(* Logix 5000 project; controller CarbonScout_MK6 vendor 1 type 14 code 154 rev 32.11; software revision 32.00; part 5 of 17 *)
(* tags used below, declared in another part *)
   Inp_OpenLS : BOOL;   // Valve Open Limit Switch 1=confirmed OPEN
   Inp_ClosedLS : BOOL;   // Valve Closed Limit Switch 1=confirmed CLOSED
   Inp_PermOK : BOOL;   // 1=Permissives OK, Valve can energize
   Inp_NBPermOK : BOOL;   // 1=Non-Bypassable Permissives OK, valve can energize
   Inp_IntlkOK : BOOL;   // 1=Interlocks OK, valve can energize
   Inp_NBIntlkOK : BOOL;   // 1=Non-Bypassable Interlocks OK, valve can energize
   Inp_IOFault : BOOL;   // Input Communication Status 0=OK, 1=fail
   Inp_Sim : BOOL;   // 1=Simulate working valve; 0=Open/Close/ Monitor actual valve
   Inp_OvrdCmd : DINT;   // Override Mode Command: 0=None, 1=Close, 2=Open
   Inp_Reset : BOOL;   // 1=Reset all fault conditions and latched Alarms
   Cfg_FailOpen : BOOL;   // 1=Fail Open (energize to close), 0=Fail Closed (energize to open)
   Cfg_HasOpenLS : BOOL;   // 1=Valve provides an Open Limit Switch signal
   Cfg_HasClosedLS : BOOL;   // 1=Valve provides a Closed Limit Switch signal
   Cfg_UseOpenLS : BOOL;   // 1=Valve Open LS should be used for failure checking
   Cfg_UseClosedLS : BOOL;   // 1=Valve Closed LS should be used for failure checking
   Cfg_LSFail : BOOL;   // 1=both switches ON=fail, 0=both switches OFF=fail
   Cfg_PCmdClear : ALIAS FOR Mode.Cfg_PCmdClear;
   Cfg_OCmdResets : BOOL;   // 1=New Oper valve cmd. resets fault, 0=reset req'd to clear fault
   Cfg_ShedOnFullStall : BOOL;   // 1=Stop Valve and Alarm on Full Stall; 0=Alarm only on Full Stall
   Cfg_ShedOnTransitStall : BOOL;   // 1=Stop Valve and Alarm on Transit Stall; 0=Alarm only on Transit Stall
   Cfg_ShedOnIOFault : BOOL;   // 1=Stop Valve and Alarm on I/O Fault; 0=Alarm only on I/O Fault
   Cfg_OvrdPermIntlk : BOOL;   // 1=Override ignores Bypassable Perm/ Intlk; 0=always use Perm/Intlk
   Cfg_SimFdbkT : DINT;   // Delay to echo back of Open/Closed status when in Simulation (sec)
   Cfg_FullStallT : DINT;   // After command, time with no motion before Fault (sec)
   Cfg_TransitStallT : DINT;   // After command, time to reach position before fault (sec)
   PSet_Owner : DINT;   // Program Owner Request ID (non-zero) or Release (zero)
   PCmd_Open : BOOL;   // Program Command to Open Valve
   PCmd_Close : BOOL;   // Program Command to Close Valve
   PCmd_Reset : BOOL;   // Program Command to Reset all Alarms requiring Reset
   PCmd_FullStallAck : ALIAS FOR FullStall.PCmd_Ack;   // Program Command to Acknowledge Full Stall Alarm
   PCmd_TransitStallAck : ALIAS FOR TransitStall.PCmd_Ack;   // Program Command to Acknowledge Transit Stall Alarm
   PCmd_IntlkTripAck : ALIAS FOR IntlkTrip.PCmd_Ack;   // Program Command to Acknowledge Interlock Trip Alarm
   PCmd_IOFaultAck : ALIAS FOR IOFault.PCmd_Ack;   // Program Command to Acknowledge I/O Fault Alarm
   OCmd_Open : BOOL;   // Operator Command to Open Valve
   OCmd_Close : BOOL;   // Operator Command to Close Valve
   OCmd_Bypass : BOOL;   // Operator Command to Bypass all Bypassable Interlocks and Permissives
   OCmd_Check : BOOL;   // Operator Command to Check (not bypass) all Interlocks and Permissives
   MCmd_Disable : BOOL;   // Maintenance Command to Disable Valve
   MCmd_Enable : BOOL;   // Maintenance Command to Enable (allow to energize) Valve
   OCmd_Reset : BOOL;   // Operator Command to Reset all Alarms requiring Reset
   OCmd_ResetAckAll : BOOL;   // Operator Command to Reset all Alarms and latched Shed conditions
   Out : BOOL;   // 1=Energize Valve Solenoid
   SrcQ_IO : DINT;   // Source and Quality of primary I/O (enumeration)
   SrcQ : DINT;   // Source and Quality of primary Val/Sts (enumeration)
   Val_Cmd : DINT;   // Device Command 0=None, 1=Close, 2=Open
   Val_Fdbk : DINT;   // Device Feedback 0=Moving, 1=Closed, 2=Opened, 3=Limit Switch Failure
   Val_Sts : DINT;   // Device Confirmed Sts 0=? 1=Closed 2=Open 5=Closing, 6=Opening, 33=Disabled
   Val_Fault : DINT;   // Device Fault Status 0=None, 16=Transit Stall, 17 = Full Stall, 32=I/O Fault, 34=Config Error
   Val_Owner : DINT;   // Current Object Owner ID (0=not owned)
   Sts_Closed : BOOL;   // 1=Valve requested to Close and is confirmed Closed
   Sts_Opening : BOOL;   // 1=Valve requested to open and awaiting open feedback
   Sts_Opened : BOOL;   // 1=Valve requested to open and is confirmed Opened
   Sts_Closing : BOOL;   // 1=Valve requested to Close and awaiting Closed feedback
   Sts_Available : BOOL;   // 1=Valve available for control by automation (Prog)
   Sts_Bypass : BOOL;   // 1=Bypassable Interlocks and Permissives are Bypassed
   Sts_BypActive : BOOL;   // 1=Bypassing Active (Bypassed or Maintenance)
   Sts_Disabled : BOOL;   // 1=Valve is Disabled
   Sts_LSFail : BOOL;   // 1=Limit Switch Overlap Failure
   Sts_NotRdy : BOOL;   // 1=Device Not Ready, see detail bits for reason
   Nrdy_Disabled : BOOL;   // 1=Device Not Ready: Device Disabled by Maintenance
   Nrdy_CfgErr : BOOL;   // 1=Device Not Ready: Configuration Error
   Nrdy_Intlk : BOOL;   // 1=Device Not Ready: Interlock Not OK
   Nrdy_Perm : BOOL;   // 1=Device Not Ready: Permissive Not OK
   Nrdy_Fail : BOOL;   // 1=Device Not Ready: Device Failure (Shed Requires Reset)
   Nrdy_IOFault : BOOL;   // 1=Device Not Ready: I/O Fault (Shed Requires Reset)
   Nrdy_NoMode : BOOL;   // 1=Device Not Ready: Device Logic Disabled / NO Mode
   Sts_MaintByp : BOOL;   // 1=A Maintenance Bypass is Active, display icon
   Sts_Err : BOOL;   // 1=Error in Config: see detail bits for reason
   Err_Timer : BOOL;   // 1=Error in Config: Invalid Check Time (use 0 to 2147483)
   Err_Sim : BOOL;   // 1=Error in Config: Invalid Simulation Time (use 0 to 2147483)
   Err_Alarm : BOOL;   // 1=Error in Config: Alarm Min On Time, Shelf Time, Severity
   Sts_Hand : ALIAS FOR Mode.Sts_Hand;
   Sts_Maint : ALIAS FOR Mode.Sts_Maint;
   Sts_Ovrd : ALIAS FOR Mode.Sts_Ovrd;
   Sts_Prog : ALIAS FOR Mode.Sts_Prog;
   Sts_Oper : ALIAS FOR Mode.Sts_Oper;
   Sts_FullStall : ALIAS FOR FullStall.Inp;   // 1=Valve Full Stall (failed to move at all)
   Sts_TransitStall : ALIAS FOR TransitStall.Inp;   // 1=Valve Transit Stall (did not reach target position)
   Sts_IntlkTrip : ALIAS FOR IntlkTrip.Inp;   // 1=Valve de-energized by an Interlock NOT OK
   Sts_IOFault : ALIAS FOR IOFault.Inp;   // I/O Comm Fault Status (0=OK, 1=Bad)
   Rdy_Open : BOOL;   // 1=Ready to receive OCmd_Open (enables HMI button)
   Rdy_Close : BOOL;   // 1=Ready to receive OCmd_Close (enables HMI button)
   Rdy_Bypass : BOOL;   // 1=Ready to receive OCmd_Bypass (enables HMI button)
   Rdy_Check : BOOL;   // 1=Ready to receive OCmd_Check (enables HMI button)
   Rdy_Disable : BOOL;   // 1=Ready to receive MCmd_Disable (enables HMI button)
   Rdy_Enable : BOOL;   // 1=Ready to receive MCmd_Enable (enables HMI button)
   P_ValveSO : BOOL;   // Unique Parameter Name for auto - discovery
   Mode : P_Mode;   // Valve Mode Selection
   IOFault : P_Alarm;   // I/O Fault Alarm
   IntlkTrip : P_Alarm;   // Interlock Trip Alarm
   TransitStall : P_Alarm;   // Valve Transit Stall (moved but did not reach target) Alarm
   FullStall : P_Alarm;   // Valve Full Stall (did not move) Alarm
   Cfg_Tag : STRING_12;   // Tagname for display on HMI
   Wrk_Open : BOOL;   // 1=Requested to OPEN Valve, 0=Requested to CLOSE Valve
   Wrk_SimOpenT : TIMER;   // Simulation Delay until Opened
   Wrk_SimCloseT : TIMER;   // Simulation Delay until Closed
   Wrk_OpenFdbk : BOOL;   // 1=LS Feedback shows valve confirmed open
   Wrk_Bypass : BOOL;   // Internal Bypassable Permissives and Interlocks are Bypassed flag
   Wrk_Disabled : BOOL;   // Internal Valve is Disabled
   Wrk_ClosedFdbk : BOOL;   // 1=LS Feedback shows valve confirmed closed
   Wrk_TransitStallT : TIMER;   // Timer for Transit Stall Check
   Wrk_FullStallT : TIMER;   // Timer for Full Stall Check
   Wrk_Sts : DINT;   // Buffer for building Val_Sts
   Wrk_SrcQ : DINT;   // Register for building Source / Quality enumeration
   Wrk_Fault : DINT;   // Buffer for building Val_Fault
   Wrk_Cmd : DINT;   // Buffer for building Val_Cmd
   Wrk_SimOpenLS : BOOL;   // Simulated valve Open Limit Switch
   Wrk_SimClosedLS : BOOL;   // Simulated valve Closed Limit Switch
   Wrk_NotRdy : BOOL;   // Device Not Ready conditions excluding shed latches
   Wrk_NoLongerSim : BOOL;   // Switched from Simulated to Real Valve this scan
   Simulation : DINT;
   test : DINT;
(* P_ValveSO, continued *)

ROUTINE Logic   (* ladder *)
// Normal Scan: control / monitor solenoid-operated valve
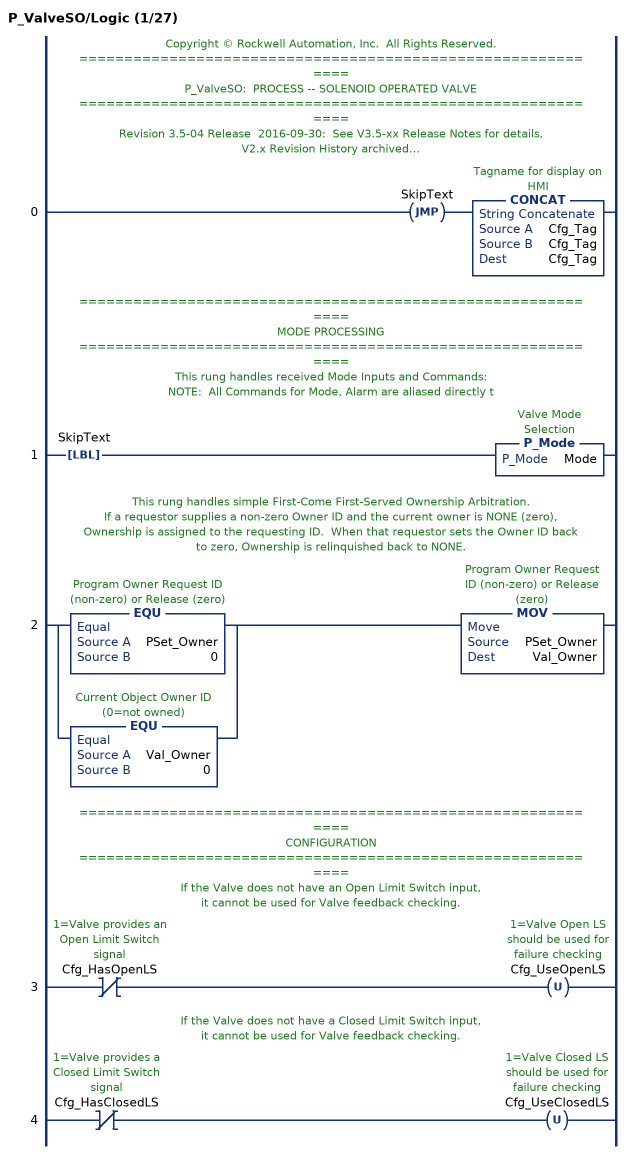
   // Copyright © Rockwell Automation, Inc.  All Rights Reserved.
   // ============================================================
   // P_ValveSO:  PROCESS -- SOLENOID OPERATED VALVE
   // ============================================================
   // Revision 3.5-04 Release  2016-09-30:  See V3.5-xx Release Notes for details.
   // V2.x Revision History archived.
   // V3.0-00  2013-06-30:  Added Inf_Lib. Using P_Alarm, P_Mode V3.0.
   // V3.0-01  2013-07-31:  Modified Parameter descriptions only.
   // V3.0-02  2013-09-03:  Modified Parameter descriptions only.
   // V3.0-03  2013-10-30:  Prescan code modified for proper powerup state.
   // Corrected Parameter descriptions and default
   // configuration values for alarms.
   // V3.0-04  2014-01-22:  Corrected Parameter Description for Val_Sts.
   // V3.1-00  2014-07-08:  Modified to use P_Alarm, P_Mode V3.1. Added Not
   // Ready reason bits (Nrdy_Xxxxx), source/quality values (SrcQ).
   // Modified to consistently use alias tag names.
   // V3.1-01  2014-09-03:  Exposed stall timers ACC/PRE (read-only). Corrections to
   // Nrdy_ trip and reset logic. Using P_Alarm, P_Mode V3.1-01.
   // V3.1-02  2014-09-30:  Unchanged, but using P_Alarm V3.1-02.
   // V3.5-01  2016-01-29:  Unchanged, but using P_Alarm V3.5.01.
   // V3.5-04  2016-09-30: Modified to align with actual device state on transition
   // from Sim to real valve.
   // ============================================================
   // This Instruction controls and monitors a single solenoid operated
   // valve (typ. two position: opened, closed) and provides:
   // *  Support for fail open (energize to close) and fail closed (energize to open, default) valves
   // *  Monitoring of limit switch feedback, display of actual valve status
   // *  Detection of failure to move (full stall), failure to reach position (transit stall)
   // *  Monitoring of Permissive conditions to allow energizing
   // *  Monitoring of Interlock conditions to de-energize
   // *  Simulation, providing feedback of a working valve while disabling outputs
   // *  Monitoring of I/O communication faults
   // *  Alarms for Full Stall, Transit Stall, Interlock Trip, I/O Fault
   // *  "Available" status for use by automation logic to know whether valve
   //       can be controlled by other objects.
   // Modes are provided by a P_Mode AOI instance.
   // Alarms are provided by P_Alarm AOI instances.
   // Modes of operation: Operator, Program, Override, Maintenance, Hand
   // ============================================================
   // SHOW LOCAL STRINGS
   // ============================================================
   // The STRINGs containing the text associated with each instance of this
   // instruction cannot be Input or Output Parameters, because STRINGs are not
   //  'atomic' types. (Inputs and Outputs must be SINT, INT, DINT, REAL, or BOOL.)
   // In order to make it easier to find and configure these STRINGs, this rung
   // was added.  THE JMP (and the LBL on the following rung)
   // MUST NOT BE REMOVED!!!
   // To view the STRINGs, go to the instruction instance (in LD or FBD), RIGHT-click
   // to bring up the context menu and select "Open Instruction Logic".
   // This rung will appear with the STRING values for the selected instance.
   // You may double-click the STRING values here to modify them as well.
   0: JMP(SkipText)CONCAT(Cfg_Tag,Cfg_Tag,Cfg_Tag);
   // ============================================================
   // MODE PROCESSING
   // ============================================================
   // This rung handles received Mode Inputs and Commands:
   // NOTE:  All Commands for Mode, Alarm are aliased directly t
   1: LBL(SkipText)P_Mode(Mode);
   // This rung handles simple First-Come First-Served Ownership Arbitration.
   // If a requestor supplies a non-zero Owner ID and the current owner is NONE (zero),
   // Ownership is assigned to the requesting ID.  When that requestor sets the Owner ID back
   // to zero, Ownership is relinquished back to NONE.
   2: [EQU(PSet_Owner,0) ,EQU(Val_Owner,0) ]MOV(PSet_Owner,Val_Owner);
   // ============================================================
   // CONFIGURATION
   // ============================================================
   // If the Valve does not have an Open Limit Switch input,
   // it cannot be used for Valve feedback checking.
   3: XIO(Cfg_HasOpenLS)OTU(Cfg_UseOpenLS);
   // If the Valve does not have a Closed Limit Switch input,
   // it cannot be used for Valve feedback checking.
   4: XIO(Cfg_HasClosedLS)OTU(Cfg_UseClosedLS);
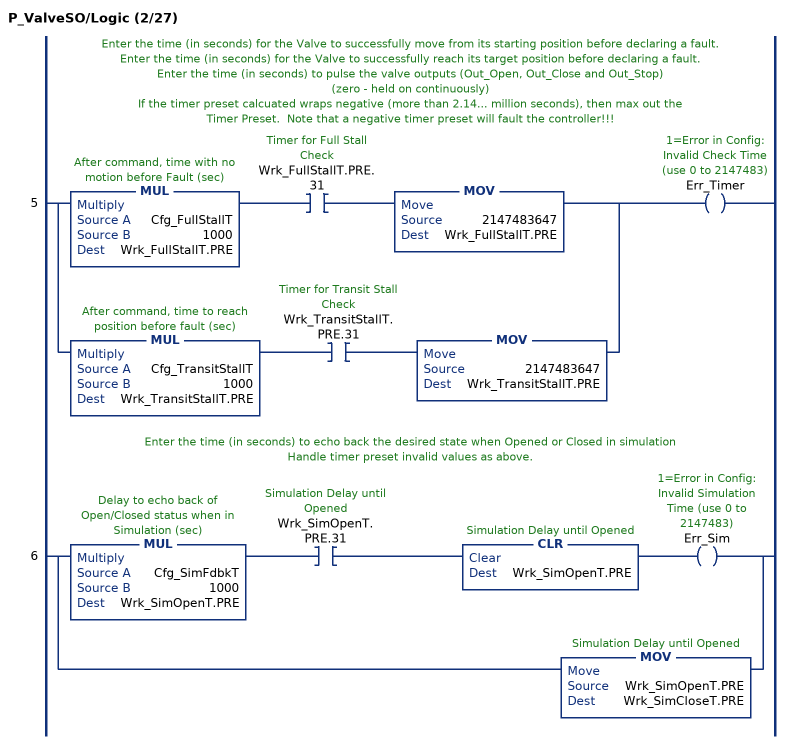
   // Enter the time (in seconds) for the Valve to successfully move from its starting position before declaring a fault.
   // Enter the time (in seconds) for the Valve to successfully reach its target position before declaring a fault.
   // Enter the time (in seconds) to pulse the valve outputs (Out_Open, Out_Close and Out_Stop)
   // (zero - held on continuously)
   // If the timer preset calcuated wraps negative (more than 2.14... million seconds), then max out the
   // Timer Preset.  Note that a negative timer preset will fault the controller!!!
   5: [MUL(Cfg_FullStallT,1000,Wrk_FullStallT.PRE) XIC(Wrk_FullStallT.PRE.31) MOV(2147483647,Wrk_FullStallT.PRE) ,MUL(Cfg_TransitStallT,1000,Wrk_TransitStallT.PRE) XIC(Wrk_TransitStallT.PRE.31) MOV(2147483647,Wrk_TransitStallT.PRE) ]OTE(Err_Timer);
   // Enter the time (in seconds) to echo back the desired state when Opened or Closed in simulation
   // Handle timer preset invalid values as above.
   6: [MUL(Cfg_SimFdbkT,1000,Wrk_SimOpenT.PRE) XIC(Wrk_SimOpenT.PRE.31) CLR(Wrk_SimOpenT.PRE) OTE(Err_Sim) ,MOV(Wrk_SimOpenT.PRE,Wrk_SimCloseT.PRE) ];
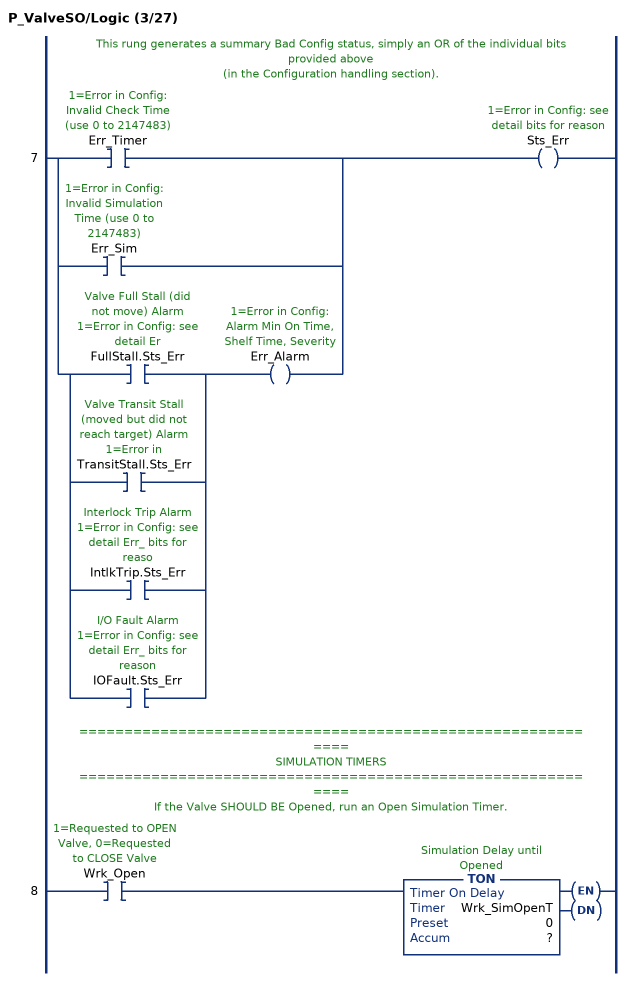
   // This rung generates a summary Bad Config status, simply an OR of the individual bits provided above
   // (in the Configuration handling section).
   7: [XIC(Err_Timer) ,XIC(Err_Sim) ,[XIC(FullStall.Sts_Err) ,XIC(TransitStall.Sts_Err) ,XIC(IntlkTrip.Sts_Err) ,XIC(IOFault.Sts_Err) ] OTE(Err_Alarm) ]OTE(Sts_Err);
   // ============================================================
   // SIMULATION TIMERS
   // ============================================================
   // If the Valve SHOULD BE Opened, run an Open Simulation Timer.
   8: XIC(Wrk_Open)TON(Wrk_SimOpenT,?,?);
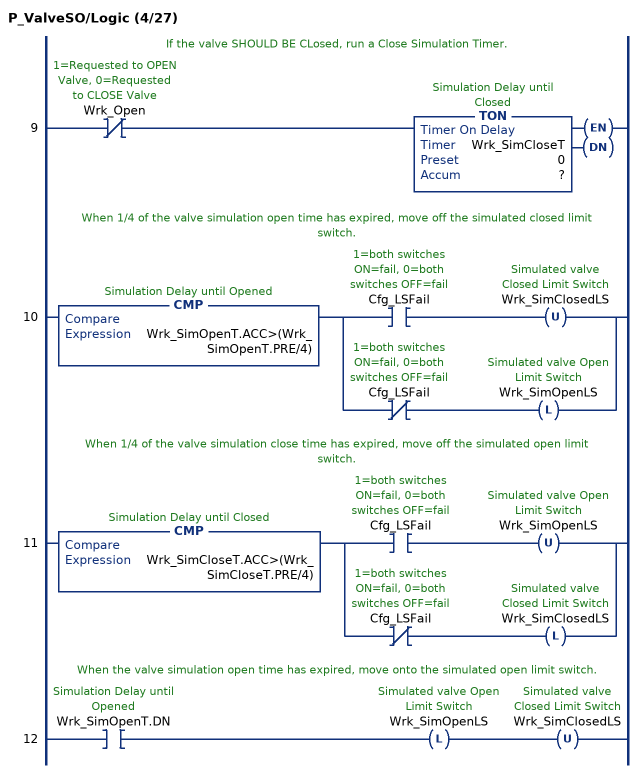
   // If the valve SHOULD BE CLosed, run a Close Simulation Timer.
   9: XIO(Wrk_Open)TON(Wrk_SimCloseT,?,?);
   // When 1/4 of the valve simulation open time has expired, move off the simulated closed limit switch.
   10: CMP(Wrk_SimOpenT.ACC>(Wrk_SimOpenT.PRE/4))[XIC(Cfg_LSFail) OTU(Wrk_SimClosedLS) ,XIO(Cfg_LSFail) OTL(Wrk_SimOpenLS) ];
   // When 1/4 of the valve simulation close time has expired, move off the simulated open limit switch.
   11: CMP(Wrk_SimCloseT.ACC>(Wrk_SimCloseT.PRE/4))[XIC(Cfg_LSFail) OTU(Wrk_SimOpenLS) ,XIO(Cfg_LSFail) OTL(Wrk_SimClosedLS) ];
   // When the valve simulation open time has expired, move onto the simulated open limit switch.
   12: XIC(Wrk_SimOpenT.DN)OTL(Wrk_SimOpenLS)OTU(Wrk_SimClosedLS);
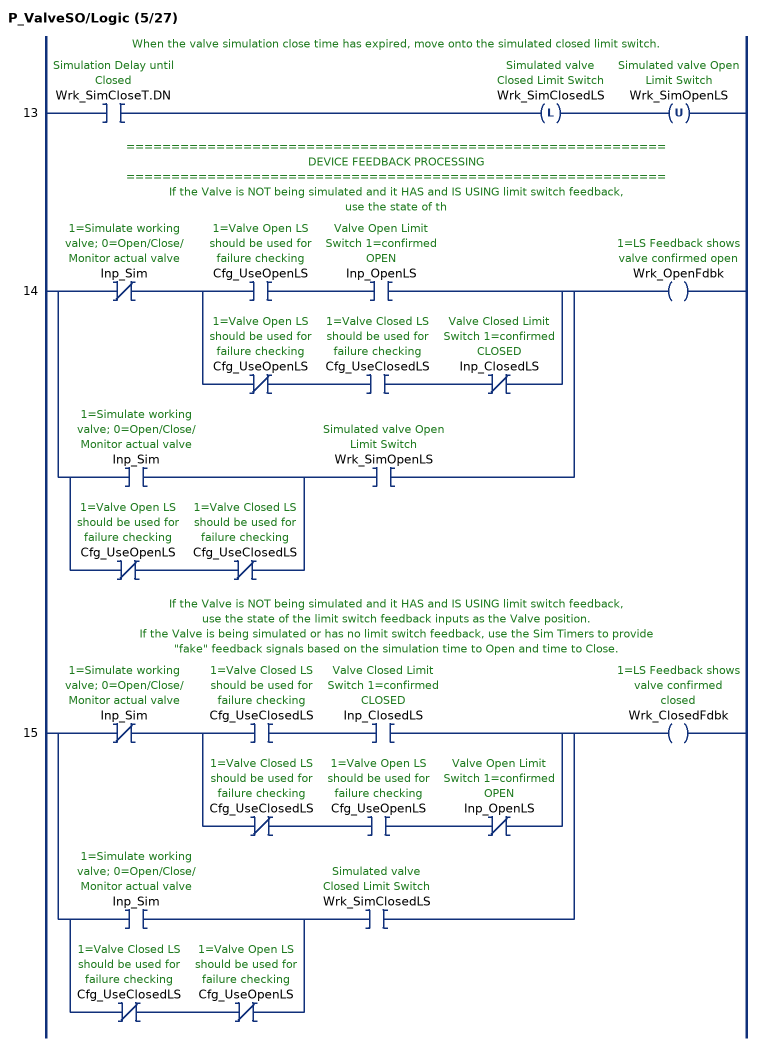
   // When the valve simulation close time has expired, move onto the simulated closed limit switch.
   13: XIC(Wrk_SimCloseT.DN)OTL(Wrk_SimClosedLS)OTU(Wrk_SimOpenLS);
   // ============================================================
   // DEVICE FEEDBACK PROCESSING
   // ============================================================
   // If the Valve is NOT being simulated and it HAS and IS USING limit switch feedback,
   // use the state of th
   14: [XIO(Inp_Sim) [XIC(Cfg_UseOpenLS) XIC(Inp_OpenLS) ,XIO(Cfg_UseOpenLS) XIC(Cfg_UseClosedLS) XIO(Inp_ClosedLS) ] ,[XIC(Inp_Sim) ,XIO(Cfg_UseOpenLS) XIO(Cfg_UseClosedLS) ] XIC(Wrk_SimOpenLS) ]OTE(Wrk_OpenFdbk);
   // If the Valve is NOT being simulated and it HAS and IS USING limit switch feedback,
   // use the state of the limit switch feedback inputs as the Valve position.
   // If the Valve is being simulated or has no limit switch feedback, use the Sim Timers to provide
   // "fake" feedback signals based on the simulation time to Open and time to Close.
   15: [XIO(Inp_Sim) [XIC(Cfg_UseClosedLS) XIC(Inp_ClosedLS) ,XIO(Cfg_UseClosedLS) XIC(Cfg_UseOpenLS) XIO(Inp_OpenLS) ] ,[XIC(Inp_Sim) ,XIO(Cfg_UseClosedLS) XIO(Cfg_UseOpenLS) ] XIC(Wrk_SimClosedLS) ]OTE(Wrk_ClosedFdbk);
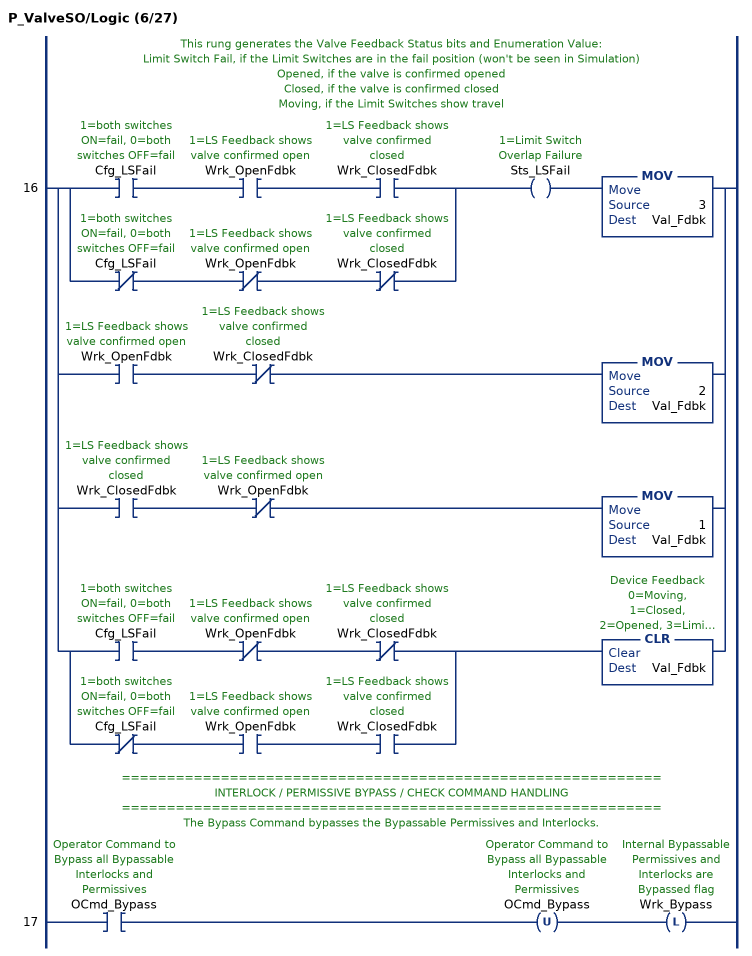
   // This rung generates the Valve Feedback Status bits and Enumeration Value:
   // Limit Switch Fail, if the Limit Switches are in the fail position (won't be seen in Simulation)
   // Opened, if the valve is confirmed opened
   // Closed, if the valve is confirmed closed
   // Moving, if the Limit Switches show travel
   16: [[XIC(Cfg_LSFail) XIC(Wrk_OpenFdbk) XIC(Wrk_ClosedFdbk) ,XIO(Cfg_LSFail) XIO(Wrk_OpenFdbk) XIO(Wrk_ClosedFdbk) ] OTE(Sts_LSFail) MOV(3,Val_Fdbk) ,XIC(Wrk_OpenFdbk) XIO(Wrk_ClosedFdbk) MOV(2,Val_Fdbk) ,XIC(Wrk_ClosedFdbk) XIO(Wrk_OpenFdbk) MOV(1,Val_Fdbk) ,[XIC(Cfg_LSFail) XIO(Wrk_OpenFdbk) XIO(Wrk_ClosedFdbk) ,XIO(Cfg_LSFail) XIC(Wrk_OpenFdbk) XIC(Wrk_ClosedFdbk) ] CLR(Val_Fdbk) ];
   // ============================================================
   // INTERLOCK / PERMISSIVE BYPASS / CHECK COMMAND HANDLING
   // ============================================================
   // The Bypass Command bypasses the Bypassable Permissives and Interlocks.
   17: XIC(OCmd_Bypass)OTU(OCmd_Bypass)OTL(Wrk_Bypass);
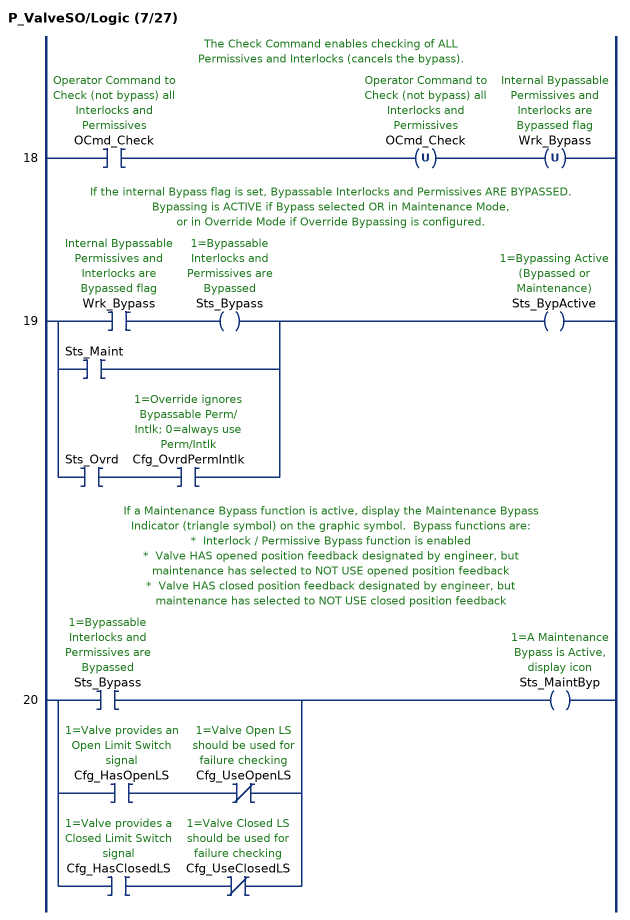
   // The Check Command enables checking of ALL
   // Permissives and Interlocks (cancels the bypass).
   18: XIC(OCmd_Check)OTU(OCmd_Check)OTU(Wrk_Bypass);
   // If the internal Bypass flag is set, Bypassable Interlocks and Permissives ARE BYPASSED.
   // Bypassing is ACTIVE if Bypass selected OR in Maintenance Mode,
   // or in Override Mode if Override Bypassing is configured.
   19: [XIC(Wrk_Bypass) OTE(Sts_Bypass) ,XIC(Sts_Maint) ,XIC(Sts_Ovrd) XIC(Cfg_OvrdPermIntlk) ]OTE(Sts_BypActive);
   // If a Maintenance Bypass function is active, display the Maintenance Bypass
   // Indicator (triangle symbol) on the graphic symbol.  Bypass functions are:
   // *  Interlock / Permissive Bypass function is enabled
   // *  Valve HAS opened position feedback designated by engineer, but
   // maintenance has selected to NOT USE opened position feedback
   // *  Valve HAS closed position feedback designated by engineer, but
   // maintenance has selected to NOT USE closed position feedback
   20: [XIC(Sts_Bypass) ,XIC(Cfg_HasOpenLS) XIO(Cfg_UseOpenLS) ,XIC(Cfg_HasClosedLS) XIO(Cfg_UseClosedLS) ]OTE(Sts_MaintByp);
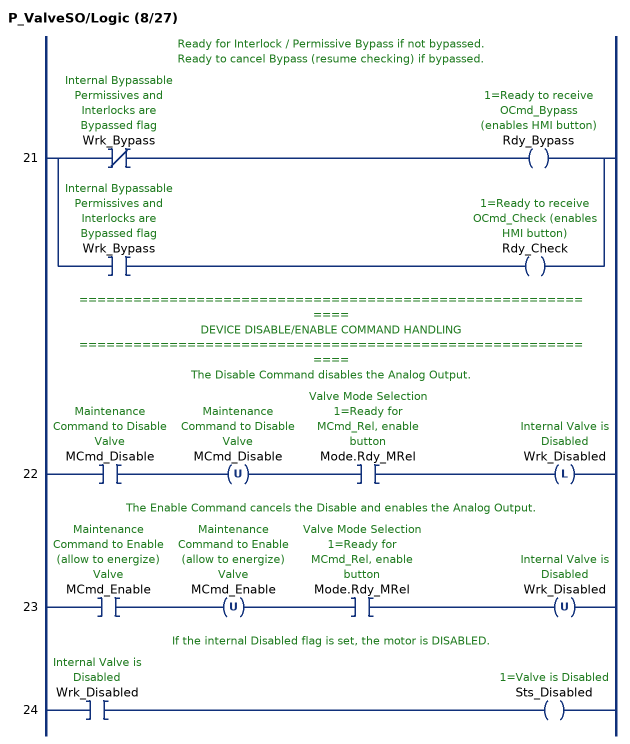
   // Ready for Interlock / Permissive Bypass if not bypassed.
   // Ready to cancel Bypass (resume checking) if bypassed.
   21: [XIO(Wrk_Bypass) OTE(Rdy_Bypass) ,XIC(Wrk_Bypass) OTE(Rdy_Check) ];
   // ============================================================
   // DEVICE DISABLE/ENABLE COMMAND HANDLING
   // ============================================================
   // The Disable Command disables the Analog Output.
   22: XIC(MCmd_Disable)OTU(MCmd_Disable)XIC(Mode.Rdy_MRel)OTL(Wrk_Disabled);
   // The Enable Command cancels the Disable and enables the Analog Output.
   23: XIC(MCmd_Enable)OTU(MCmd_Enable)XIC(Mode.Rdy_MRel)OTU(Wrk_Disabled);
   // If the internal Disabled flag is set, the motor is DISABLED.
   24: XIC(Wrk_Disabled)OTE(Sts_Disabled);
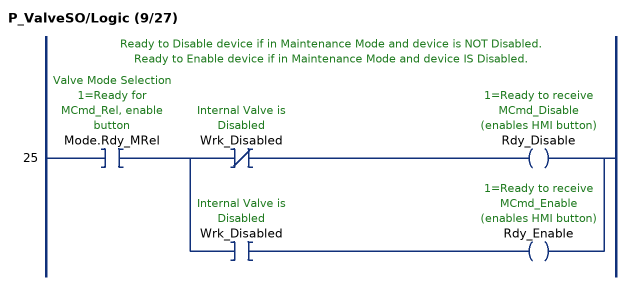
   // Ready to Disable device if in Maintenance Mode and device is NOT Disabled.
   // Ready to Enable device if in Maintenance Mode and device IS Disabled.
   25: XIC(Mode.Rdy_MRel)[XIO(Wrk_Disabled) OTE(Rdy_Disable) ,XIC(Wrk_Disabled) OTE(Rdy_Enable) ];
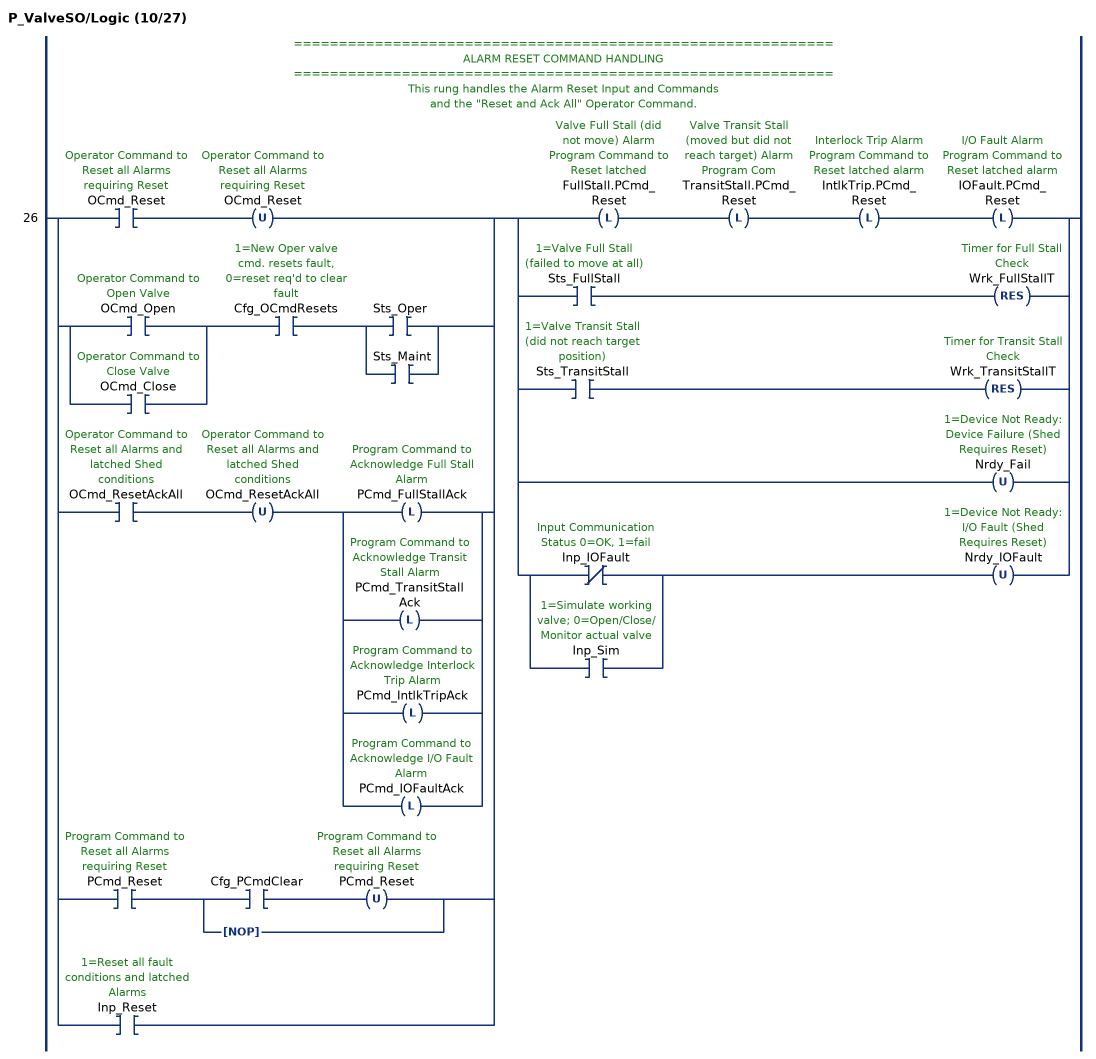
   // ============================================================
   // ALARM RESET COMMAND HANDLING
   // ============================================================
   // This rung handles the Alarm Reset Input and Commands
   // and the "Reset and Ack All" Operator Command.
   26: [XIC(OCmd_Reset) OTU(OCmd_Reset) ,[XIC(OCmd_Open) ,XIC(OCmd_Close) ] XIC(Cfg_OCmdResets) [XIC(Sts_Oper) ,XIC(Sts_Maint) ] ,XIC(OCmd_ResetAckAll) OTU(OCmd_ResetAckAll) [OTL(PCmd_FullStallAck) ,OTL(PCmd_TransitStallAck) ,OTL(PCmd_IntlkTripAck) ,OTL(PCmd_IOFaultAck) ] ,XIC(PCmd_Reset) [XIC(Cfg_PCmdClear) OTU(PCmd_Reset) ,NOP() ] ,XIC(Inp_Reset) ][OTL(FullStall.PCmd_Reset) OTL(TransitStall.PCmd_Reset) OTL(IntlkTrip.PCmd_Reset) OTL(IOFault.PCmd_Reset) ,XIC(Sts_FullStall) RES(Wrk_FullStallT) ,XIC(Sts_TransitStall) RES(Wrk_TransitStallT) ,OTU(Nrdy_Fail) ,[XIO(Inp_IOFault) ,XIC(Inp_Sim) ] OTU(Nrdy_IOFault) ];
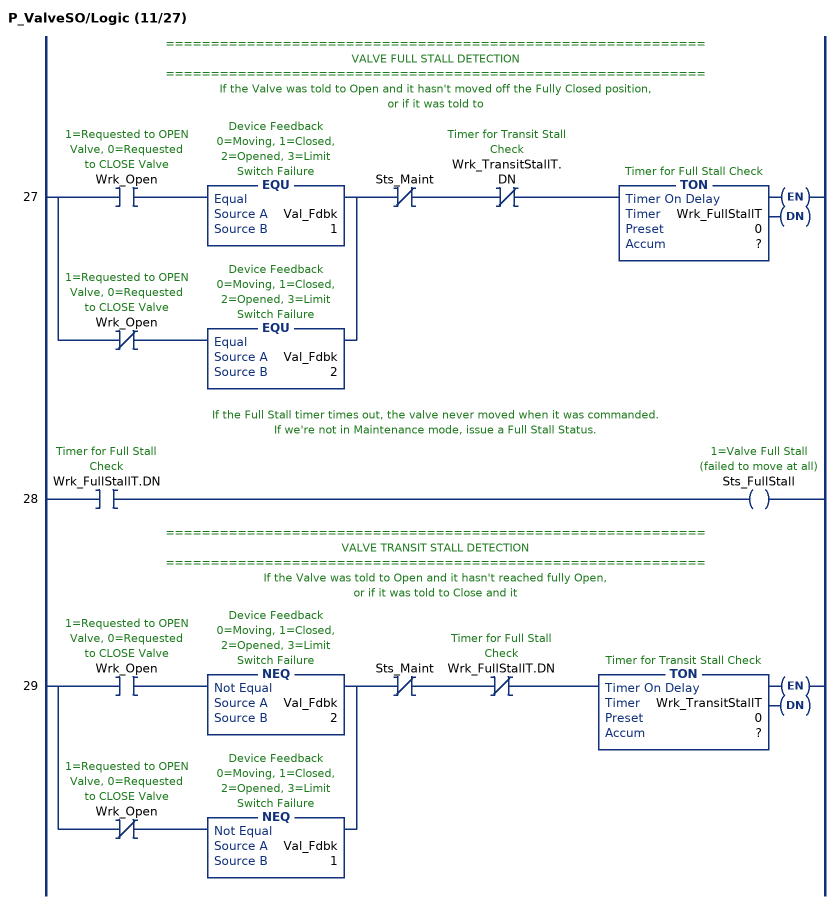
   // ============================================================
   // VALVE FULL STALL DETECTION
   // ============================================================
   // If the Valve was told to Open and it hasn't moved off the Fully Closed position,
   // or if it was told to
   27: [XIC(Wrk_Open) EQU(Val_Fdbk,1) ,XIO(Wrk_Open) EQU(Val_Fdbk,2) ]XIO(Sts_Maint)XIO(Wrk_TransitStallT.DN)TON(Wrk_FullStallT,?,?);
   // If the Full Stall timer times out, the valve never moved when it was commanded.
   // If we're not in Maintenance mode, issue a Full Stall Status.
   28: XIC(Wrk_FullStallT.DN)OTE(Sts_FullStall);
   // ============================================================
   // VALVE TRANSIT STALL DETECTION
   // ============================================================
   // If the Valve was told to Open and it hasn't reached fully Open,
   // or if it was told to Close and it
   29: [XIC(Wrk_Open) NEQ(Val_Fdbk,2) ,XIO(Wrk_Open) NEQ(Val_Fdbk,1) ]XIO(Sts_Maint)XIO(Wrk_FullStallT.DN)TON(Wrk_TransitStallT,?,?);
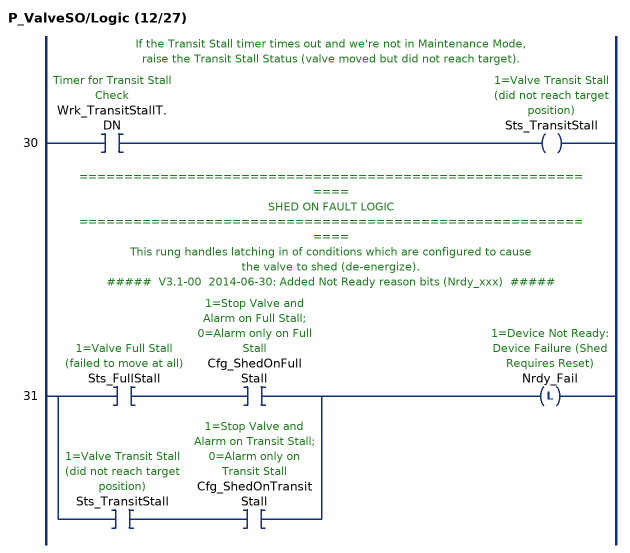
   // If the Transit Stall timer times out and we're not in Maintenance Mode,
   // raise the Transit Stall Status (valve moved but did not reach target).
   30: XIC(Wrk_TransitStallT.DN)OTE(Sts_TransitStall);
   // ============================================================
   // SHED ON FAULT LOGIC
   // ============================================================
   // This rung handles latching in of conditions which are configured to cause
   // the valve to shed (de-energize).
   // #####  V3.1-00  2014-06-30: Added Not Ready reason bits (Nrdy_xxx)  #####
   31: [XIC(Sts_FullStall) XIC(Cfg_ShedOnFullStall) ,XIC(Sts_TransitStall) XIC(Cfg_ShedOnTransitStall) ]OTL(Nrdy_Fail);
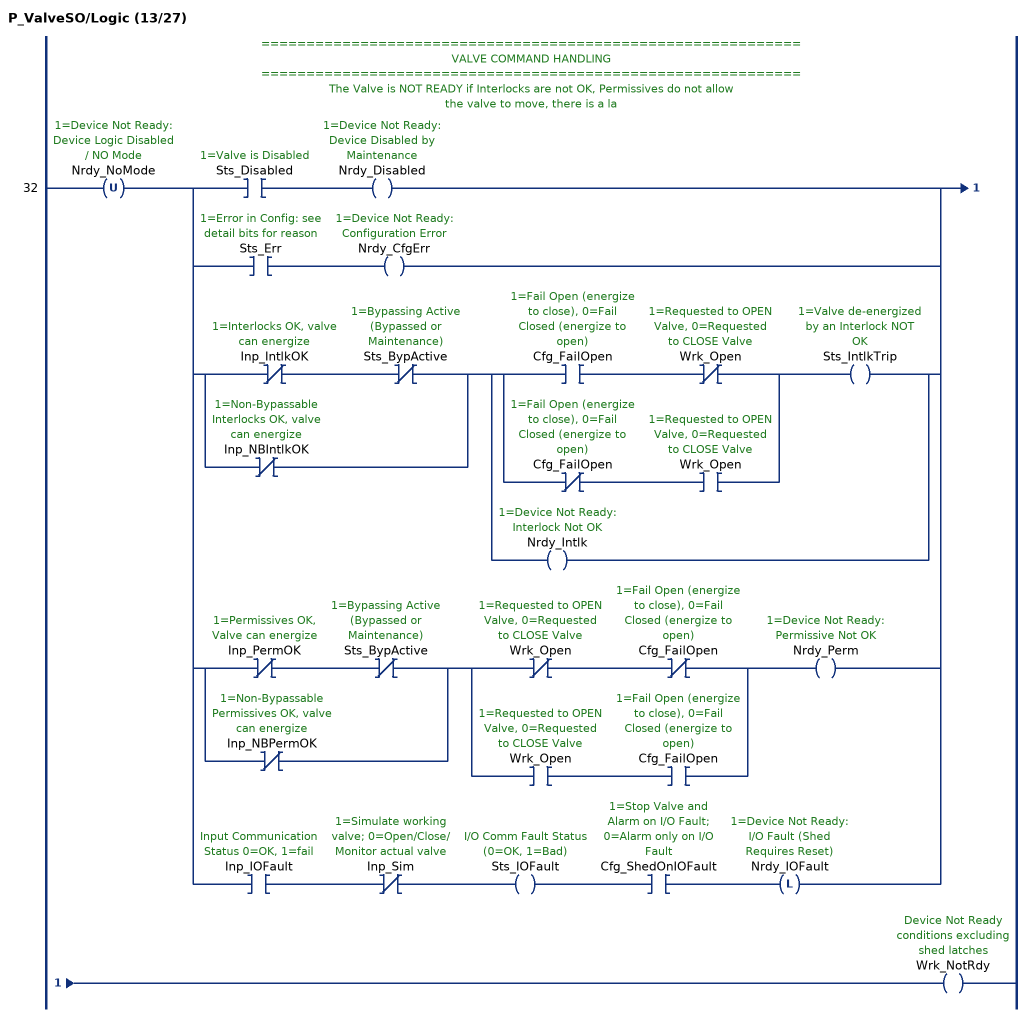
   // ============================================================
   // VALVE COMMAND HANDLING
   // ============================================================
   // The Valve is NOT READY if Interlocks are not OK, Permissives do not allow
   // the valve to move, there is a la
   32: OTU(Nrdy_NoMode)[XIC(Sts_Disabled) OTE(Nrdy_Disabled) ,XIC(Sts_Err) OTE(Nrdy_CfgErr) ,[XIO(Inp_IntlkOK) XIO(Sts_BypActive) ,XIO(Inp_NBIntlkOK) ] [[XIC(Cfg_FailOpen) XIO(Wrk_Open) ,XIO(Cfg_FailOpen) XIC(Wrk_Open) ] OTE(Sts_IntlkTrip) ,OTE(Nrdy_Intlk) ] ,[XIO(Inp_PermOK) XIO(Sts_BypActive) ,XIO(Inp_NBPermOK) ] [XIO(Wrk_Open) XIO(Cfg_FailOpen) ,XIC(Wrk_Open) XIC(Cfg_FailOpen) ] OTE(Nrdy_Perm) ,XIC(Inp_IOFault) XIO(Inp_Sim) OTE(Sts_IOFault) XIC(Cfg_ShedOnIOFault) OTL(Nrdy_IOFault) ]OTE(Wrk_NotRdy);
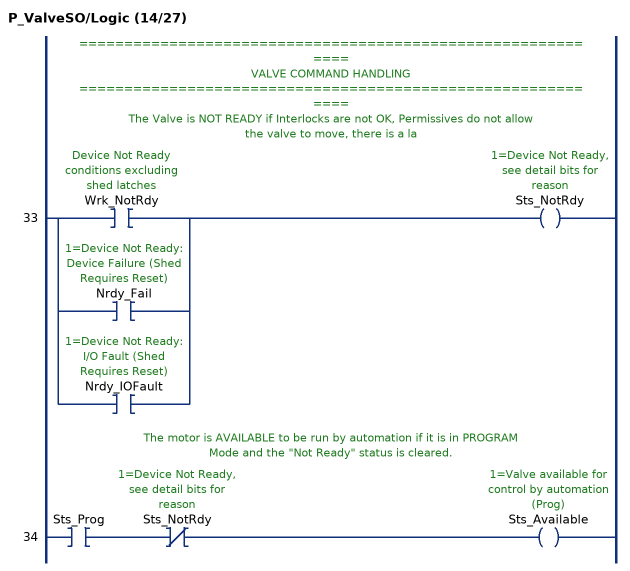
   // ============================================================
   // VALVE COMMAND HANDLING
   // ============================================================
   // The Valve is NOT READY if Interlocks are not OK, Permissives do not allow
   // the valve to move, there is a la
   33: [XIC(Wrk_NotRdy) ,XIC(Nrdy_Fail) ,XIC(Nrdy_IOFault) ]OTE(Sts_NotRdy);
   // The motor is AVAILABLE to be run by automation if it is in PROGRAM
   // Mode and the "Not Ready" status is cleared.
   34: XIC(Sts_Prog)XIO(Sts_NotRdy)OTE(Sts_Available);
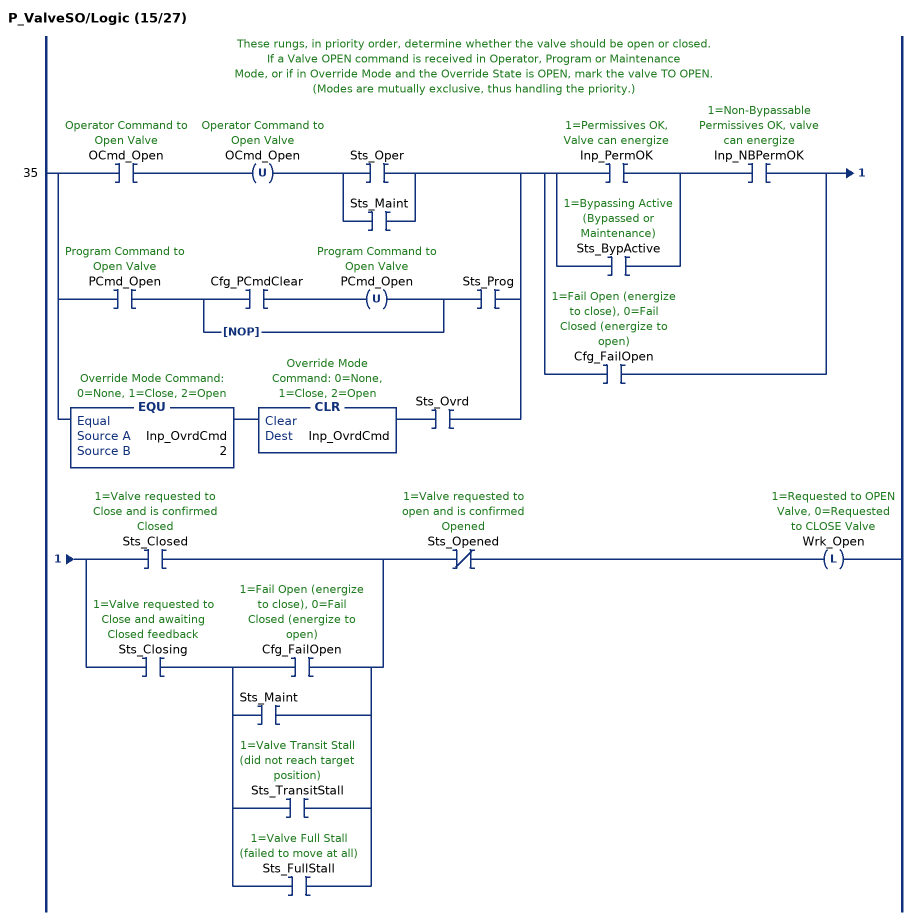
   // These rungs, in priority order, determine whether the valve should be open or closed.
   // If a Valve OPEN command is received in Operator, Program or Maintenance
   // Mode, or if in Override Mode and the Override State is OPEN, mark the valve TO OPEN.
   // (Modes are mutually exclusive, thus handling the priority.)
   35: [XIC(OCmd_Open) OTU(OCmd_Open) [XIC(Sts_Oper) ,XIC(Sts_Maint) ] ,XIC(PCmd_Open) [XIC(Cfg_PCmdClear) OTU(PCmd_Open) ,NOP() ] XIC(Sts_Prog) ,EQU(Inp_OvrdCmd,2) CLR(Inp_OvrdCmd) XIC(Sts_Ovrd) ][[XIC(Inp_PermOK) ,XIC(Sts_BypActive) ] XIC(Inp_NBPermOK) ,XIC(Cfg_FailOpen) ][XIC(Sts_Closed) ,XIC(Sts_Closing) [XIC(Cfg_FailOpen) ,XIC(Sts_Maint) ,XIC(Sts_TransitStall) ,XIC(Sts_FullStall) ] ]XIO(Sts_Opened)OTL(Wrk_Open);
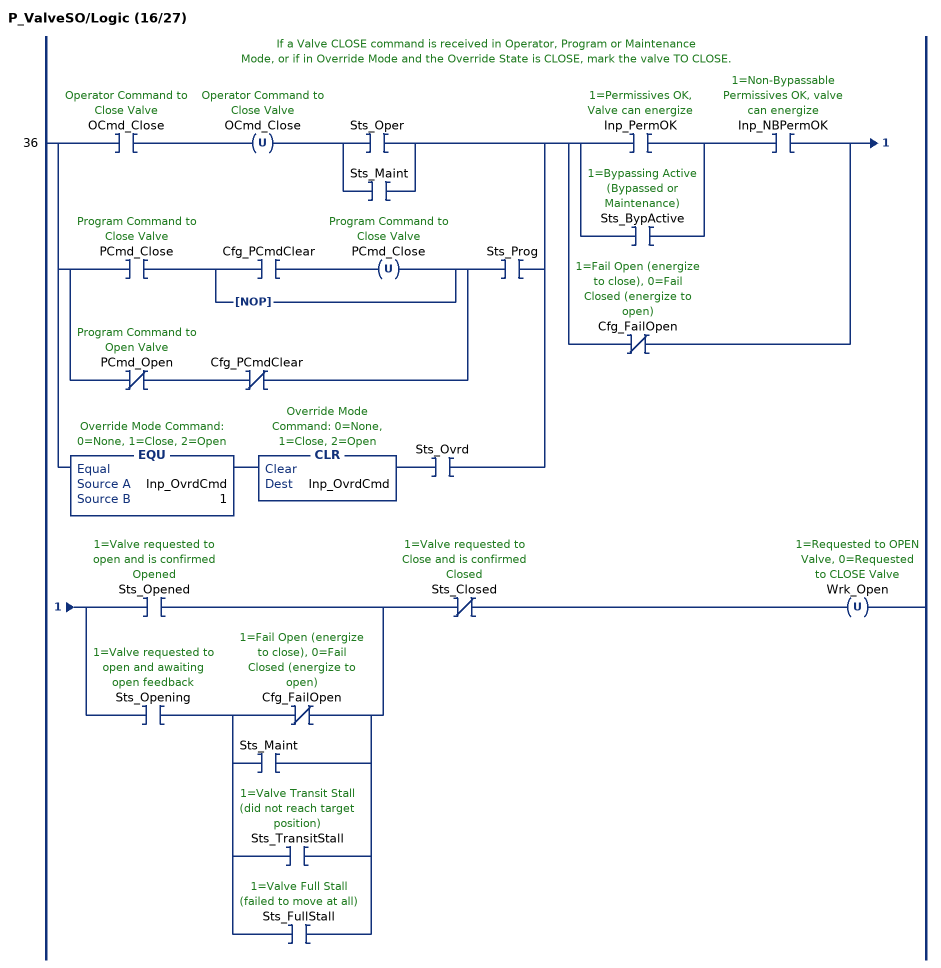
   // If a Valve CLOSE command is received in Operator, Program or Maintenance
   // Mode, or if in Override Mode and the Override State is CLOSE, mark the valve TO CLOSE.
   36: [XIC(OCmd_Close) OTU(OCmd_Close) [XIC(Sts_Oper) ,XIC(Sts_Maint) ] ,[XIC(PCmd_Close) [XIC(Cfg_PCmdClear) OTU(PCmd_Close) ,NOP() ] ,XIO(PCmd_Open) XIO(Cfg_PCmdClear) ] XIC(Sts_Prog) ,EQU(Inp_OvrdCmd,1) CLR(Inp_OvrdCmd) XIC(Sts_Ovrd) ][[XIC(Inp_PermOK) ,XIC(Sts_BypActive) ] XIC(Inp_NBPermOK) ,XIO(Cfg_FailOpen) ][XIC(Sts_Opened) ,XIC(Sts_Opening) [XIO(Cfg_FailOpen) ,XIC(Sts_Maint) ,XIC(Sts_TransitStall) ,XIC(Sts_FullStall) ] ]XIO(Sts_Closed)OTU(Wrk_Open);
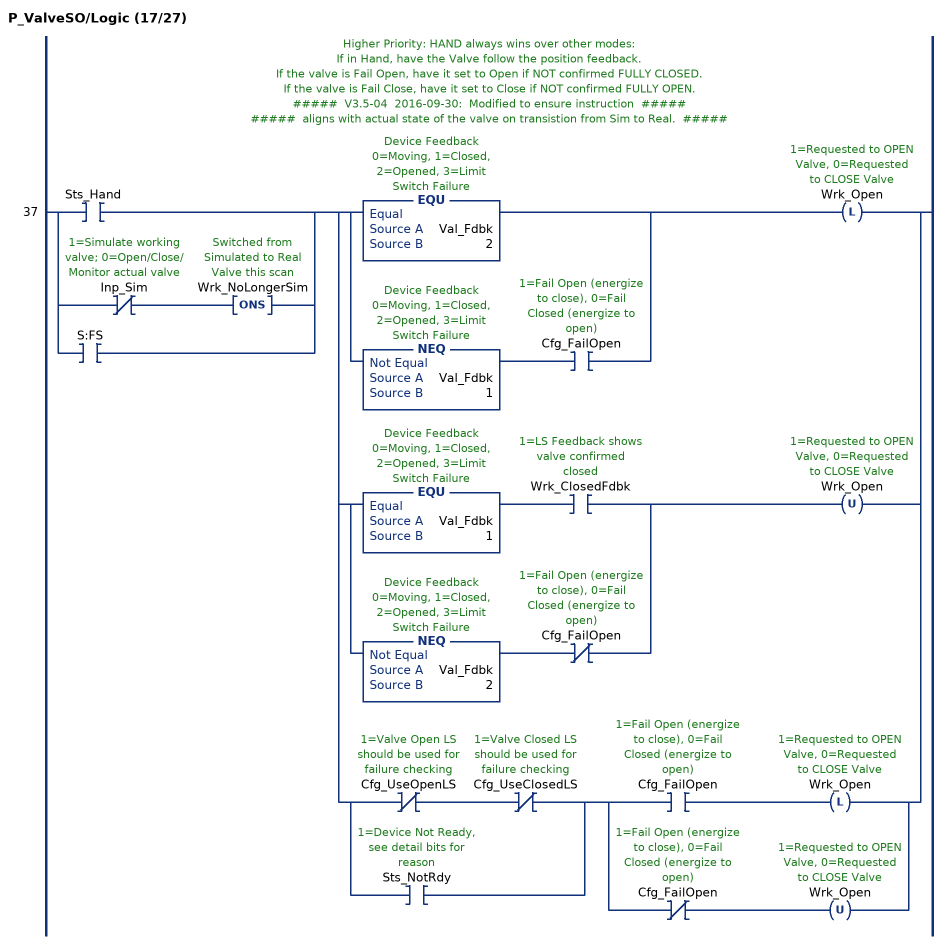
   // Higher Priority: HAND always wins over other modes:
   // If in Hand, have the Valve follow the position feedback.
   // If the valve is Fail Open, have it set to Open if NOT confirmed FULLY CLOSED.
   // If the valve is Fail Close, have it set to Close if NOT confirmed FULLY OPEN.
   // #####  V3.5-04  2016-09-30:  Modified to ensure instruction  #####
   // #####  aligns with actual state of the valve on transistion from Sim to Real.  #####
   37: [XIC(Sts_Hand) ,XIO(Inp_Sim) ONS(Wrk_NoLongerSim) ,XIC(S:FS) ][[EQU(Val_Fdbk,2) ,NEQ(Val_Fdbk,1) XIC(Cfg_FailOpen) ] OTL(Wrk_Open) ,[EQU(Val_Fdbk,1) XIC(Wrk_ClosedFdbk) ,NEQ(Val_Fdbk,2) XIO(Cfg_FailOpen) ] OTU(Wrk_Open) ,[XIO(Cfg_UseOpenLS) XIO(Cfg_UseClosedLS) ,XIC(Sts_NotRdy) ] [XIC(Cfg_FailOpen) OTL(Wrk_Open) ,XIO(Cfg_FailOpen) OTU(Wrk_Open) ] ];
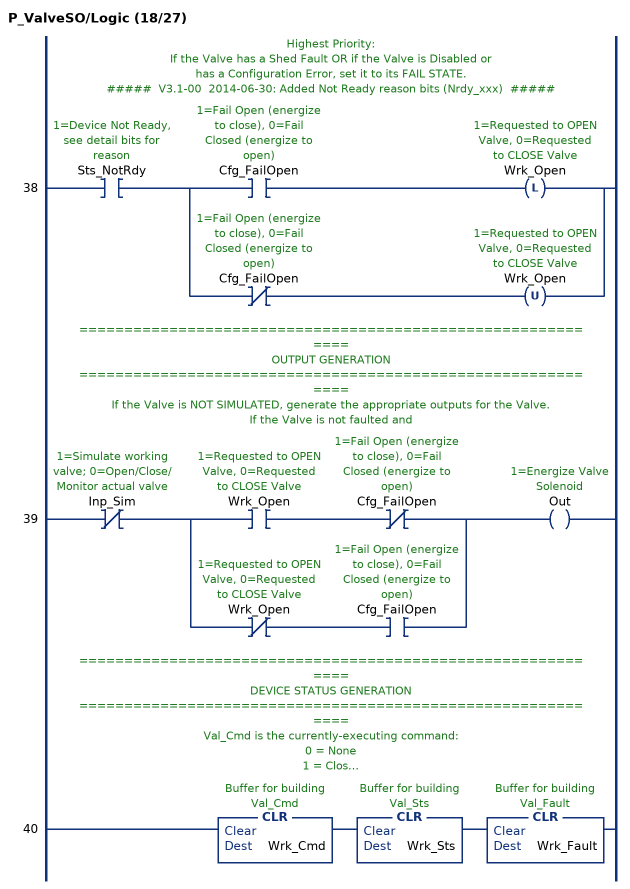
   // Highest Priority:
   // If the Valve has a Shed Fault OR if the Valve is Disabled or
   // has a Configuration Error, set it to its FAIL STATE.
   // #####  V3.1-00  2014-06-30: Added Not Ready reason bits (Nrdy_xxx)  #####
   38: XIC(Sts_NotRdy)[XIC(Cfg_FailOpen) OTL(Wrk_Open) ,XIO(Cfg_FailOpen) OTU(Wrk_Open) ];
   // ============================================================
   // OUTPUT GENERATION
   // ============================================================
   // If the Valve is NOT SIMULATED, generate the appropriate outputs for the Valve.
   // If the Valve is not faulted and
   39: XIO(Inp_Sim)[XIC(Wrk_Open) XIO(Cfg_FailOpen) ,XIO(Wrk_Open) XIC(Cfg_FailOpen) ]OTE(Out);
   // ============================================================
   // DEVICE STATUS GENERATION
   // ============================================================
   // Val_Cmd is the currently-executing command:
   // 0 = None
   // 1 = Close
   // 2 = Open
   // Val_Sts is the current devi
   40: CLR(Wrk_Cmd)CLR(Wrk_Sts)CLR(Wrk_Fault);
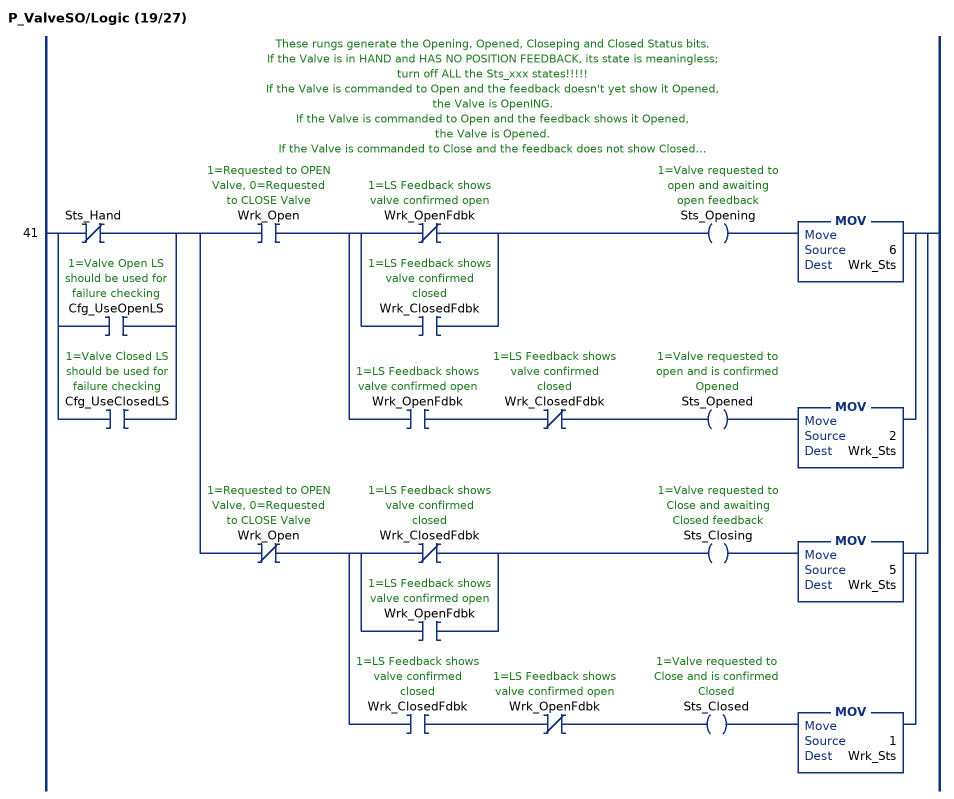
   // These rungs generate the Opening, Opened, Closeping and Closed Status bits.
   // If the Valve is in HAND and HAS NO POSITION FEEDBACK, its state is meaningless;
   // turn off ALL the Sts_xxx states!!!!!
   // If the Valve is commanded to Open and the feedback doesn't yet show it Opened,
   // the Valve is OpenING.
   // If the Valve is commanded to Open and the feedback shows it Opened,
   // the Valve is Opened.
   // If the Valve is commanded to Close and the feedback does not show Closed,
   // the Valve is CloseING.
   // If the Valve is commanded to Close and the feedback shows it has Closed,
   // the Valve is Closed.
   41: [XIO(Sts_Hand) ,XIC(Cfg_UseOpenLS) ,XIC(Cfg_UseClosedLS) ][XIC(Wrk_Open) [[XIO(Wrk_OpenFdbk) ,XIC(Wrk_ClosedFdbk) ] OTE(Sts_Opening) MOV(6,Wrk_Sts) ,XIC(Wrk_OpenFdbk) XIO(Wrk_ClosedFdbk) OTE(Sts_Opened) MOV(2,Wrk_Sts) ] ,XIO(Wrk_Open) [[XIO(Wrk_ClosedFdbk) ,XIC(Wrk_OpenFdbk) ] OTE(Sts_Closing) MOV(5,Wrk_Sts) ,XIC(Wrk_ClosedFdbk) XIO(Wrk_OpenFdbk) OTE(Sts_Closed) MOV(1,Wrk_Sts) ] ];
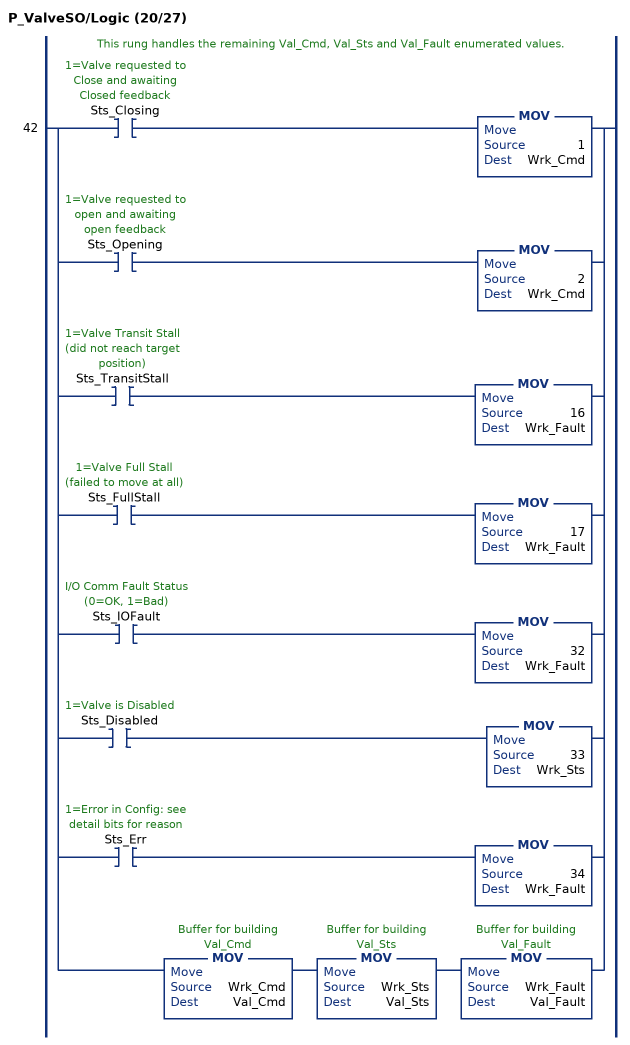
   // This rung handles the remaining Val_Cmd, Val_Sts and Val_Fault enumerated values.
   42: [XIC(Sts_Closing) MOV(1,Wrk_Cmd) ,XIC(Sts_Opening) MOV(2,Wrk_Cmd) ,XIC(Sts_TransitStall) MOV(16,Wrk_Fault) ,XIC(Sts_FullStall) MOV(17,Wrk_Fault) ,XIC(Sts_IOFault) MOV(32,Wrk_Fault) ,XIC(Sts_Disabled) MOV(33,Wrk_Sts) ,XIC(Sts_Err) MOV(34,Wrk_Fault) ,MOV(Wrk_Cmd,Val_Cmd) MOV(Wrk_Sts,Val_Sts) MOV(Wrk_Fault,Val_Fault) ];
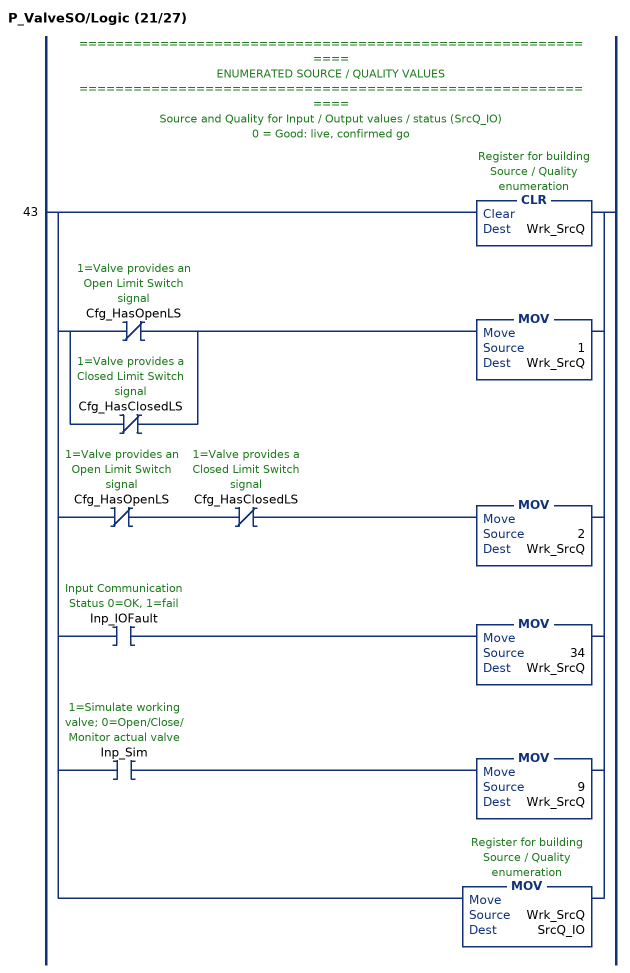
   // ============================================================
   // ENUMERATED SOURCE / QUALITY VALUES
   // ============================================================
   // Source and Quality for Input / Output values / status (SrcQ_IO)
   // 0 = Good: live, confirmed go
   43: [CLR(Wrk_SrcQ) ,[XIO(Cfg_HasOpenLS) ,XIO(Cfg_HasClosedLS) ] MOV(1,Wrk_SrcQ) ,XIO(Cfg_HasOpenLS) XIO(Cfg_HasClosedLS) MOV(2,Wrk_SrcQ) ,XIC(Inp_IOFault) MOV(34,Wrk_SrcQ) ,XIC(Inp_Sim) MOV(9,Wrk_SrcQ) ,MOV(Wrk_SrcQ,SrcQ_IO) ];
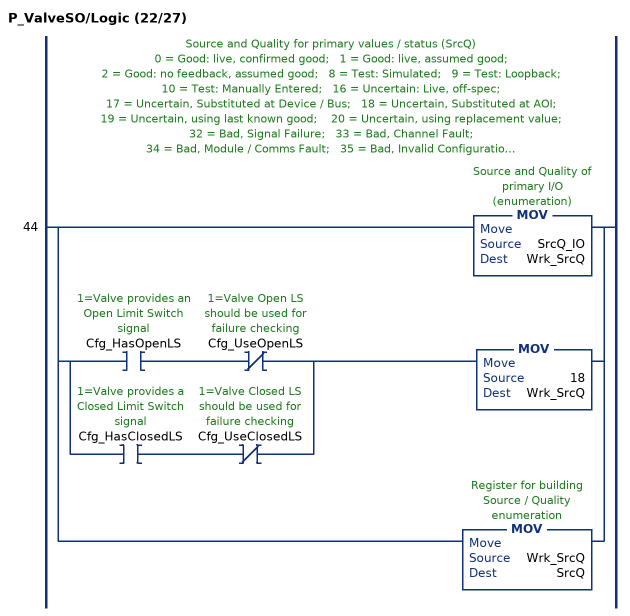
   // Source and Quality for primary values / status (SrcQ)
   // 0 = Good: live, confirmed good;   1 = Good: live, assumed good;
   // 2 = Good: no feedback, assumed good;   8 = Test: Simulated;   9 = Test: Loopback;
   // 10 = Test: Manually Entered;   16 = Uncertain: Live, off-spec;
   // 17 = Uncertain, Substituted at Device / Bus;   18 = Uncertain, Substituted at AOI;
   // 19 = Uncertain, using last known good;    20 = Uncertain, using replacement value;
   // 32 = Bad, Signal Failure;   33 = Bad, Channel Fault;
   // 34 = Bad, Module / Comms Fault;   35 = Bad, Invalid Configuration
   // #####  V3.1-00  2014-06-30:  Added rung for Source/Quality enumerations.  #####
   44: [MOV(SrcQ_IO,Wrk_SrcQ) ,[XIC(Cfg_HasOpenLS) XIO(Cfg_UseOpenLS) ,XIC(Cfg_HasClosedLS) XIO(Cfg_UseClosedLS) ] MOV(18,Wrk_SrcQ) ,MOV(Wrk_SrcQ,SrcQ) ];
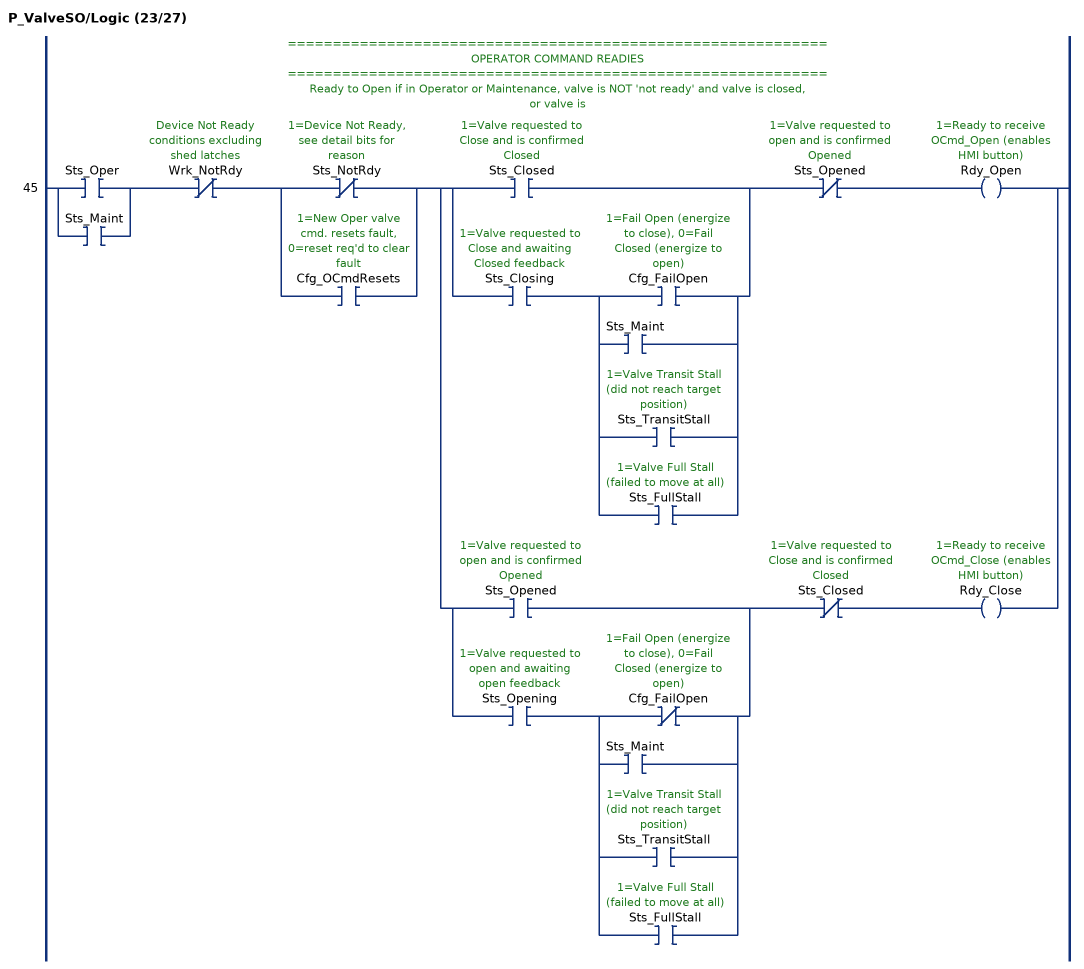
   // ============================================================
   // OPERATOR COMMAND READIES
   // ============================================================
   // Ready to Open if in Operator or Maintenance, valve is NOT 'not ready' and valve is closed,
   // or valve is
   45: [XIC(Sts_Oper) ,XIC(Sts_Maint) ]XIO(Wrk_NotRdy)[XIO(Sts_NotRdy) ,XIC(Cfg_OCmdResets) ][[XIC(Sts_Closed) ,XIC(Sts_Closing) [XIC(Cfg_FailOpen) ,XIC(Sts_Maint) ,XIC(Sts_TransitStall) ,XIC(Sts_FullStall) ] ] XIO(Sts_Opened) OTE(Rdy_Open) ,[XIC(Sts_Opened) ,XIC(Sts_Opening) [XIO(Cfg_FailOpen) ,XIC(Sts_Maint) ,XIC(Sts_TransitStall) ,XIC(Sts_FullStall) ] ] XIO(Sts_Closed) OTE(Rdy_Close) ];
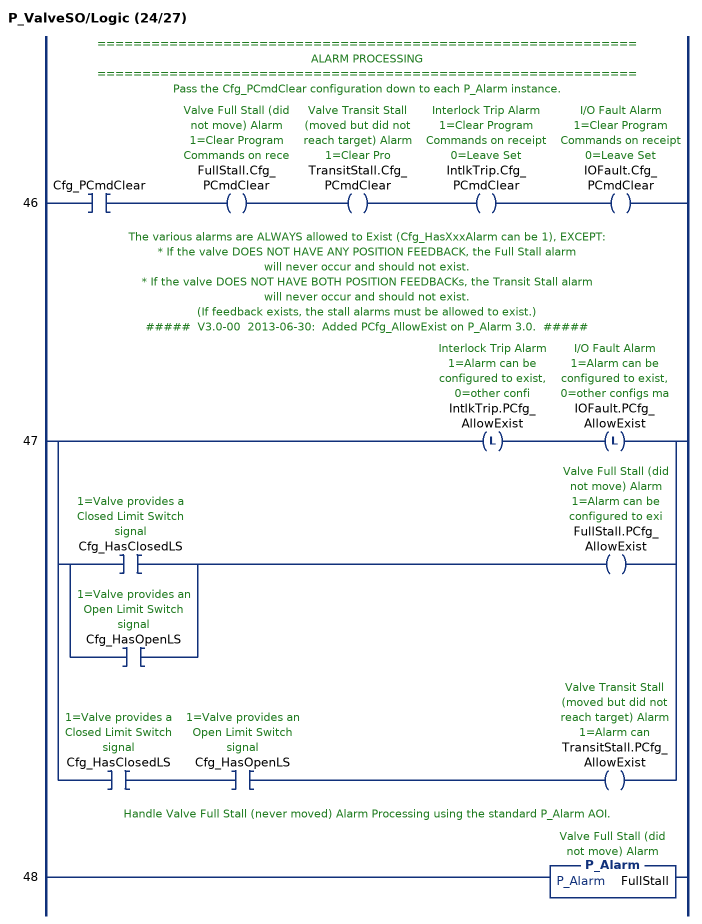
   // ============================================================
   // ALARM PROCESSING
   // ============================================================
   // Pass the Cfg_PCmdClear configuration down to each P_Alarm instance.
   46: XIC(Cfg_PCmdClear)OTE(FullStall.Cfg_PCmdClear)OTE(TransitStall.Cfg_PCmdClear)OTE(IntlkTrip.Cfg_PCmdClear)OTE(IOFault.Cfg_PCmdClear);
   // The various alarms are ALWAYS allowed to Exist (Cfg_HasXxxAlarm can be 1), EXCEPT:
   // * If the valve DOES NOT HAVE ANY POSITION FEEDBACK, the Full Stall alarm
   // will never occur and should not exist.
   // * If the valve DOES NOT HAVE BOTH POSITION FEEDBACKs, the Transit Stall alarm
   // will never occur and should not exist.
   // (If feedback exists, the stall alarms must be allowed to exist.)
   // #####  V3.0-00  2013-06-30:  Added PCfg_AllowExist on P_Alarm 3.0.  #####
   47: [OTL(IntlkTrip.PCfg_AllowExist) OTL(IOFault.PCfg_AllowExist) ,[XIC(Cfg_HasClosedLS) ,XIC(Cfg_HasOpenLS) ] OTE(FullStall.PCfg_AllowExist) ,XIC(Cfg_HasClosedLS) XIC(Cfg_HasOpenLS) OTE(TransitStall.PCfg_AllowExist) ];
   // Handle Valve Full Stall (never moved) Alarm Processing using the standard P_Alarm AOI.
   48: P_Alarm(FullStall);
